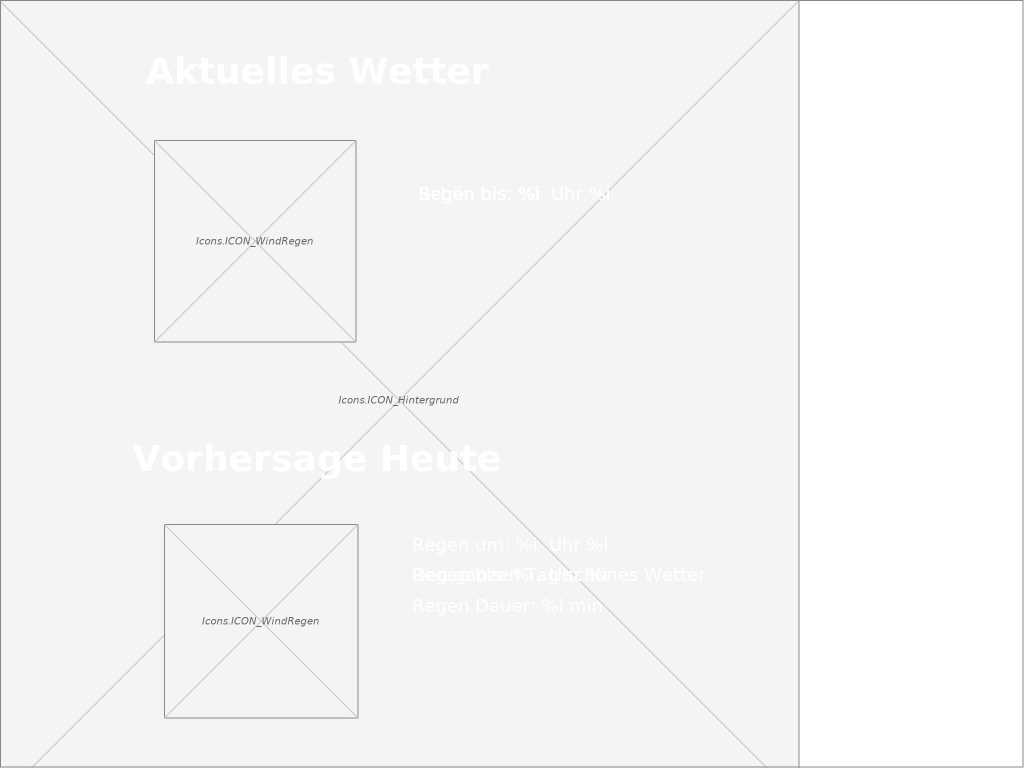
VISUALIZATION Wetterbericht  // 1024x768
    Image (-1,0 800x800), image: Icons.ICON_Hintergrund
    Image (154,140 202x202), image: Icons.ICON_WindRegen
        p84334746: Wetterbericht_Bild
    Label (121,56 393x30), "Aktuelles Wetter"
    Label (121,430 392x57), "Vorhersage Heute"
    Image (164,524 194x194), image: Icons.ICON_WindRegen
        p84334746: Wetterbericht_Vorhersage_Bild
    Textfield (409,530 231x30), "Regen um: %i", text variable: Regen_Stunde, invisible if: NOT Rege_Heute
    Textfield (546,530 231x30), "Uhr %i", text variable: Regen_Minute, invisible if: NOT Rege_Heute
    Textfield (409,560 231x30), "Regen bis: %i", text variable: Regen_Stunde_Ende, invisible if: NOT Rege_Heute
    Textfield (546,560 231x30), "Uhr %i", text variable: Regen_Minute_Ende, invisible if: NOT Rege_Heute
    Textfield (409,591 231x30), "Regen Dauer: %i min", text variable: Regen_Dauer, invisible if: NOT Rege_Heute
    Textfield (364,179 231x30), "Regen bis: %i", text variable: Regen_Stunde_Ende, invisible if: NOT Regen
    Textfield (548,179 231x30), "Uhr %i", text variable: Regen_Minute_Ende, invisible if: NOT Regen
    Textfield (364,179 231x30), "Schön bis: %i", text variable: Regen_Stunde, invisible if: NOT Rege_Heute OR Regen
    Textfield (548,179 231x30), "Uhr %i", text variable: Regen_Minute, invisible if: NOT Rege_Heute OR Regen
    Textfield (409,560 352x30), "Den ganzen Tag schönes Wetter", text variable: Regen_Stunde, invisible if: Rege_Heute
END_VISUALIZATION

(* stored: Version 1.1.0.1, ProductVersion 3.1.4018.5
   Visu Wetterbericht: Id {3904a983-2bea-4375-b192-54e0be994497} *)
